(* CoDeSys 2.3 export: INC_TO_AMPERE.EXP *)

(* POU Line Communication/Single Line/Helper/INC_TO_AMPERE, ST *)
FUNCTION INC_TO_AMPERE : REAL
VAR_INPUT
	IN		:	WORD;
END_VAR
(* calculation from increments to ampere *)
INC_TO_AMPERE := (80.0 		(* max. current *)
                                       / 29126)	(* -> 32767 - 3641  Increments of the module for MAX_CURRENT *)
						* WORD_TO_INT(IN);
END_FUNCTION
